// TIA Portal V16 export
// export: Created 2022-02-04T14:40:18.7822852Z, ExportSetting WithDefaults, DisplayName Totally Integrated Automation Portal, DisplayVersion V16 Update 1, DisplayName TIA Portal Version Control Interface, DisplayVersion V16, DisplayName TIA Portal Openness, DisplayVersion V16, DisplayName SINAMICS Startdrive Advanced, DisplayVersion V16 Update 5, DisplayName SINAMICS Startdrive G130, G150, S120, S150, SINAMICS MV, S210, DisplayVersion V16 Update 5, DisplayName SINAMICS Startdrive G110M, G120, G120C, G120D, G120P, G115D, DisplayVersion V16 Update 5, DisplayName STEP 7 Professional, DisplayVersion V16, DisplayName STEP 7 Safety, DisplayVersion V16, DisplayName WinCC Advanced, DisplayVersion V16, DisplayName SIMATIC Visualization Architect, DisplayVersion V16
DATA_BLOCK "ALG"   // DB9
VERSION : 0.1
// stored: AutoNumber true, IsOnlyStoredInLoadMemory false, IsWriteProtectedInAS false
   VAR RETAIN
      Ready_defect : Bool;
      Alarm_defect : Bool;
      Auto_defect : Bool;
      Ready_loading : Bool;
      Alarm_loading : Bool;
      Auto_loading : Bool;
      Ready_Sorting : Bool;
      Alarm_Sorting : Bool;
      Auto_Sorting : Bool;
      Ready_Gasket : Bool;
      Alarm_Gasket : Bool;
      Auto_Gasket : Bool;
      Ready_Rout : Bool;
      Alarm_Rout : Bool;
      Auto_Rout : Bool;
      Reset : Bool;
      start_encoder : Bool := true;   // начать счет энкодера
      reset_encoder : Bool;   // направление влево
      ForceFinishMainPFM : Bool;
      ForceFinishPFMDefect : Bool;
      DefectivePacketIsPushed : Bool;
      PacketReadyRollOut : Bool;   // пакет готов к отгрузке
      EmptyLodems : Bool;
      AddGasketLayer : Bool;   // добавить слой прокладок
      ConfirmGasketsBrak : Bool;   // бит подтверждения на слой брака
      ModeChang : Bool;
      STOP : Bool;   // глобальный тсоп
      VirtualAuto : Bool;
      RampSyncSig : Bool;
      HELPER : Bool;
      TestCounter : Int;
      TestCounter2 : Int;
      LayerVolume : DInt;   // текущий объем пакета
      Volume : DInt;
      Meandr : Int;   // счет для меандра
      PermMovM323 : Time;   // тайминг на работу упоров
      SqueezeRamp : Time := T#1ms;   // задержка на движение рамы
      SqueezeUporPFM : Time;
   END_VAR
BEGIN
END_DATA_BLOCK
